INTERFACE PUBLIC UnholdingCommands EXTENDS RunningStateCommands, ActionStateCommands, HoldableStateCommands

END_INTERFACE

(* stored: Version 1.1.0.1, ProductVersion 3.1.4026.18
   Itf UnholdingCommands: Id {2ed69181-4160-0c5d-1d9d-bb7c14caa326} *)
